DATA_BLOCK "MOD"   // DB57
// stored: InstanceOfName AFB_MODULES, InstanceOfType FB
"AFB_MODULES"
BEGIN
   ADIN[0].input := 536.3774;
   ADIN[0].monitorfault := TRUE;
   ADIN[0].p1s := FALSE;
   ADIN[0].p100ms := TRUE;
   ADIN[0].generalackn := FALSE;
   ADIN[0].reset := FALSE;
   ADIN[0].mute := FALSE;
   ADIN[0].Unit := WSTRING#'';
   ADIN[0].Switch := FALSE;
   ADIN[0].alarm_adin := FALSE;
   ADIN[0].plcackn_adin := FALSE;
   ADIN[0].siren_adin := FALSE;
   ADIN[0].hmiackn_adin := FALSE;
   ADIN[0].i."time".on_set := 0;
   ADIN[0].i."time".off_set := 0;
   ADIN[0].i."time".on_act := 0;
   ADIN[0].i."time".off_act := 0;
   ADIN[0].i.setup.comparison := 0;
   ADIN[0].i.setup.reference := 1900.0;
   ADIN[0].i.setup.alarm := FALSE;
   ADIN[0].i.setup.triggerversion := FALSE;
   ADIN[0].i.faults.adin.setup.en := FALSE;
   ADIN[0].i.faults.adin.setup.spon := 0.0;
   ADIN[0].i.faults.adin.don.countup := FALSE;
   ADIN[0].i.faults.adin.don.sp := 0;
   ADIN[0].i.faults.adin.don.actual := 0;
   ADIN[0].i.faults.adin.don.end := FALSE;
   ADIN[0].i.faults.adin.status.plcackn := FALSE;
   ADIN[0].i.faults.adin.status.alarm := FALSE;
   ADIN[0].i.faults.adin.status.siren := FALSE;
   ADIN[0].i.faults.fpreset := FALSE;
   ADIN[0].i.sim.cmdon := FALSE;
   ADIN[0].i.sim.cmdoff := FALSE;
   ADIN[0].i.sim.simulated := FALSE;
   ADIN[0].i.sim.cmdforce := FALSE;
   ADIN[0].i.sim.cmdunforce := FALSE;
   ADIN[0].i.sim.forced := FALSE;
   ADIN[0].i.status.rawinput := 525.5537;
   ADIN[0].i.status.processed := FALSE;
   ADIN[0].i.status.switch_active := FALSE;
   ADIN[0].i.status.alarm_monitor := FALSE;
   ADIN[0].i.status.fault := FALSE;
   ADIN[0].i.unit := WSTRING#'';
   // AIN[0] : LT44_01_01
   AIN[0].in := 12542;
   AIN[0].generalackn := FALSE;
   AIN[0].reset := FALSE;
   AIN[0].mute := FALSE;
   AIN[0].p1s := FALSE;
   AIN[0].p100ms := FALSE;
   AIN[0].t_sys := DTL#2025-10-07-08:40:00.150809;
   AIN[0]."type" := 2;
   AIN[0].output := 4.536314;
   AIN[0].i.chn."type" := 1;
   AIN[0].i.chn.in := 12534.0;
   AIN[0].i.chn.high := 27648.0;
   AIN[0].i.chn.low := 0.0;
   AIN[0].i.scale.high := 10.0;
   AIN[0].i.scale.low := 0.0;
   AIN[0].i.scale.factor := 1.0;
   AIN[0].i.scale.set := TRUE;
   AIN[0].i.sim.en := FALSE;
   AIN[0].i.sim.value := 0.0;
   AIN[0].i.exp.en := FALSE;
   AIN[0].i.exp.init := FALSE;
   AIN[0].i.exp.T := 0.0;
   AIN[0].i.exp.limit := 0.0;
   AIN[0].i.exp."dt" := 0.0;
   AIN[0].i.exp."a" := 0.0;
   AIN[0].i.faults.hh.setup.en := TRUE;
   AIN[0].i.faults.hh.setup.spon := 1.0;
   AIN[0].i.faults.hh.don.countup := FALSE;
   AIN[0].i.faults.hh.don.sp := 10;
   AIN[0].i.faults.hh.don.actual := 0;
   AIN[0].i.faults.hh.don.end := FALSE;
   AIN[0].i.faults.hh.status.plcackn := FALSE;
   AIN[0].i.faults.hh.status.alarm := FALSE;
   AIN[0].i.faults.hh.status.siren := FALSE;
   AIN[0].i.faults.h.setup.en := TRUE;
   AIN[0].i.faults.h.setup.spon := 10.0;
   AIN[0].i.faults.h.don.countup := FALSE;
   AIN[0].i.faults.h.don.sp := 100;
   AIN[0].i.faults.h.don.actual := 0;
   AIN[0].i.faults.h.don.end := FALSE;
   AIN[0].i.faults.h.status.plcackn := FALSE;
   AIN[0].i.faults.h.status.alarm := FALSE;
   AIN[0].i.faults.h.status.siren := FALSE;
   AIN[0].i.faults.l.setup.en := TRUE;
   AIN[0].i.faults.l.setup.spon := 0.0;
   AIN[0].i.faults.l.don.countup := FALSE;
   AIN[0].i.faults.l.don.sp := 0;
   AIN[0].i.faults.l.don.actual := 0;
   AIN[0].i.faults.l.don.end := FALSE;
   AIN[0].i.faults.l.status.plcackn := FALSE;
   AIN[0].i.faults.l.status.alarm := FALSE;
   AIN[0].i.faults.l.status.siren := FALSE;
   AIN[0].i.faults.ll.setup.en := TRUE;
   AIN[0].i.faults.ll.setup.spon := 0.0;
   AIN[0].i.faults.ll.don.countup := FALSE;
   AIN[0].i.faults.ll.don.sp := 0;
   AIN[0].i.faults.ll.don.actual := 0;
   AIN[0].i.faults.ll.don.end := FALSE;
   AIN[0].i.faults.ll.status.plcackn := FALSE;
   AIN[0].i.faults.ll.status.alarm := FALSE;
   AIN[0].i.faults.ll.status.siren := FALSE;
   AIN[0].i.faults.sp_hh := 5.6;
   AIN[0].i.faults.sp_h := 5.3;
   AIN[0].i.faults.sp_l := 0.5;
   AIN[0].i.faults.sp_ll := 0.2;
   AIN[0].i.faults.fpreset := FALSE;
   AIN[0].i.trendlow := -1.0;
   AIN[0].i.trendhigh := 12.0;
   AIN[0].i.scaled := 4.53342;
   AIN[0].i.output := 4.53342;
   AIN[0].i.unit := WSTRING#'m';
   AIN[0].exp.init := FALSE;
   AIN[0].exp.Sn := 4.536314;
   AIN[0].exp.Xn := 4.536314;
   AIN[0].exp.lim_up := 0.0;
   AIN[0].exp.lim_down := 0.0;
   AIN[0].exp.t_buf := DTL#2025-10-07-08:40:00.150809;
   AIN[0].exp.t_diff := FALSE;
   AIN[0].calc.scalespan := 10.0;
   AIN[0].calc.chnspan := 27648.0;
   AIN[0].calc.xmax := 27648.0;
   AIN[0].calc.xmin := 0.0;
   AIN[0].calc.ymax := 10.0;
   AIN[0].calc.ymin := 0.0;
   AIN[0].calc.x := 12542.0;
   AIN[0].calc.y := 4.536314;
   AIN[0].calc.sign := TRUE;
   AIN[0].calc.scale."type" := 0;
   AIN[0].calc.scale.in := 0.0;
   AIN[0].calc.scale.scalehigh := 0.0;
   AIN[0].calc.scale.scalelow := 0.0;
   AIN[0].calc.scale.channelhigh := 0.0;
   AIN[0].calc.scale.channellow := 0.0;
   AIN[0].calc.scale.factor := 0.0;
   AIN[0].calc.scale.calc1 := 0.0;
   AIN[0].calc.scale.span := 0.0;
   AIN[0].calc.scale.output := 0.0;
   AIN[0].lastob_si.EV_CLASS := 16#00;
   AIN[0].lastob_si.EV_NUM := 16#00;
   AIN[0].lastob_si.PRIORITY := 16#00;
   AIN[0].lastob_si.NUM := 16#00;
   AIN[0].lastob_si.TYP2_3 := 16#00;
   AIN[0].lastob_si.TYP1 := 16#00;
   AIN[0].lastob_si.ZI1 := 16#0000;
   AIN[0].lastob_si.ZI2_3 := 16#0000_0000;
   AIN[0].startob_si.EV_CLASS := 16#00;
   AIN[0].startob_si.EV_NUM := 16#00;
   AIN[0].startob_si.PRIORITY := 16#00;
   AIN[0].startob_si.NUM := 16#00;
   AIN[0].startob_si.TYP2_3 := 16#00;
   AIN[0].startob_si.TYP1 := 16#00;
   AIN[0].startob_si.ZI1 := 16#0000;
   AIN[0].startob_si.ZI2_3 := 16#0000_0000;
   AIN[0].err := 0;
   AIN[0].hilow := TRUE;
   AIN[0].factor := FALSE;
   DIFF[0].Minuend := 0.0;
   DIFF[0].Subtrahend := 0.0;
   DIFF[0].unit := WSTRING#'';
   DIFF[0].generalackn := FALSE;
   DIFF[0].reset := FALSE;
   DIFF[0].mute := FALSE;
   DIFF[0].p1s := FALSE;
   DIFF[0].p100ms := FALSE;
   DIFF[0].output := 0.0;
   DIFF[0].i.sim.en := FALSE;
   DIFF[0].i.sim.value := 0.0;
   DIFF[0].i.faults.hh.setup.en := FALSE;
   DIFF[0].i.faults.hh.setup.spon := 0.0;
   DIFF[0].i.faults.hh.don.countup := FALSE;
   DIFF[0].i.faults.hh.don.sp := 0;
   DIFF[0].i.faults.hh.don.actual := 0;
   DIFF[0].i.faults.hh.don.end := FALSE;
   DIFF[0].i.faults.hh.status.plcackn := FALSE;
   DIFF[0].i.faults.hh.status.alarm := FALSE;
   DIFF[0].i.faults.hh.status.siren := FALSE;
   DIFF[0].i.faults.h.setup.en := FALSE;
   DIFF[0].i.faults.h.setup.spon := 0.0;
   DIFF[0].i.faults.h.don.countup := FALSE;
   DIFF[0].i.faults.h.don.sp := 0;
   DIFF[0].i.faults.h.don.actual := 0;
   DIFF[0].i.faults.h.don.end := FALSE;
   DIFF[0].i.faults.h.status.plcackn := FALSE;
   DIFF[0].i.faults.h.status.alarm := FALSE;
   DIFF[0].i.faults.h.status.siren := FALSE;
   DIFF[0].i.faults.l.setup.en := FALSE;
   DIFF[0].i.faults.l.setup.spon := 0.0;
   DIFF[0].i.faults.l.don.countup := FALSE;
   DIFF[0].i.faults.l.don.sp := 0;
   DIFF[0].i.faults.l.don.actual := 0;
   DIFF[0].i.faults.l.don.end := FALSE;
   DIFF[0].i.faults.l.status.plcackn := FALSE;
   DIFF[0].i.faults.l.status.alarm := FALSE;
   DIFF[0].i.faults.l.status.siren := FALSE;
   DIFF[0].i.faults.ll.setup.en := FALSE;
   DIFF[0].i.faults.ll.setup.spon := 0.0;
   DIFF[0].i.faults.ll.don.countup := FALSE;
   DIFF[0].i.faults.ll.don.sp := 0;
   DIFF[0].i.faults.ll.don.actual := 0;
   DIFF[0].i.faults.ll.don.end := FALSE;
   DIFF[0].i.faults.ll.status.plcackn := FALSE;
   DIFF[0].i.faults.ll.status.alarm := FALSE;
   DIFF[0].i.faults.ll.status.siren := FALSE;
   DIFF[0].i.faults.sp_hh := 0.0;
   DIFF[0].i.faults.sp_h := 0.0;
   DIFF[0].i.faults.sp_l := 0.0;
   DIFF[0].i.faults.sp_ll := 0.0;
   DIFF[0].i.faults.fpreset := FALSE;
   DIFF[0].i.minuend := 0.0;
   DIFF[0].i.subtrahend := 0.0;
   DIFF[0].i.trendhigh := 0.0;
   DIFF[0].i.output := 0.0;
   DIFF[0].i.unit := WSTRING#'';
   // DIN[0] : LsH44_01_01
   DIN[0].input := TRUE;
   DIN[0].monitorfault := TRUE;
   DIN[0].p1s := FALSE;
   DIN[0].p100ms := FALSE;
   DIN[0].generalackn := FALSE;
   DIN[0].reset := FALSE;
   DIN[0].mute := FALSE;
   DIN[0].Switch := FALSE;
   DIN[0].alarm_din := FALSE;
   DIN[0].plcackn_din := FALSE;
   DIN[0].siren_din := FALSE;
   DIN[0].hmiackn_din := FALSE;
   DIN[0].i."time".on_set := 0;
   DIN[0].i."time".off_set := 0;
   DIN[0].i."time".on_act := 0;
   DIN[0].i."time".off_act := 0;
   DIN[0].i.setup.polarity := TRUE;
   DIN[0].i.setup.triggerversion := FALSE;
   DIN[0].i.faults.din.setup.en := FALSE;
   DIN[0].i.faults.din.setup.spon := 0.0;
   DIN[0].i.faults.din.don.countup := FALSE;
   DIN[0].i.faults.din.don.sp := 0;
   DIN[0].i.faults.din.don.actual := 0;
   DIN[0].i.faults.din.don.end := FALSE;
   DIN[0].i.faults.din.status.plcackn := FALSE;
   DIN[0].i.faults.din.status.alarm := FALSE;
   DIN[0].i.faults.din.status.siren := FALSE;
   DIN[0].i.faults.fpreset := FALSE;
   DIN[0].i.sim.cmdon := FALSE;
   DIN[0].i.sim.cmdoff := FALSE;
   DIN[0].i.sim.simulated := FALSE;
   DIN[0].i.sim.cmdforce := FALSE;
   DIN[0].i.sim.cmdunforce := FALSE;
   DIN[0].i.sim.forced := FALSE;
   DIN[0].i.status.rawinput := TRUE;
   DIN[0].i.status.processed := FALSE;
   DIN[0].i.status.switch_active := FALSE;
   DIN[0].i.status.alarm_monitor := FALSE;
   DIN[0].i.status.fault := FALSE;
   // MTR[0] : P44_05
   MTR[0].start := FALSE;
   MTR[0].spsource := FALSE;
   MTR[0].followup := FALSE;
   MTR[0].pidrun := TRUE;
   MTR[0].fb := FALSE;
   MTR[0].mcb := FALSE;
   MTR[0].ctrl := TRUE;
   MTR[0].vfdnotrip := FALSE;
   MTR[0].block := FALSE;
   MTR[0].generalackn := FALSE;
   MTR[0].reset := FALSE;
   MTR[0].mute := FALSE;
   MTR[0].autoset := FALSE;
   MTR[0].manualset := FALSE;
   MTR[0].p1s := FALSE;
   MTR[0].p100ms := FALSE;
   MTR[0].blink := TRUE;
   MTR[0].PV := 4.000289;
   MTR[0].PV_unit := WSTRING#'';
   MTR[0].EXT_SP := 0.0;
   MTR[0].FUP := 20.0;
   MTR[0].Out_unit := WSTRING#'';
   MTR[0].run := FALSE;
   MTR[0].vfb := FALSE;
   MTR[0].reference := 0;
   MTR[0].i.cmd.auto := FALSE;
   MTR[0].i.cmd.man := FALSE;
   MTR[0].i.cmd.start := FALSE;
   MTR[0].i.cmd.stop := FALSE;
   MTR[0].i.ind.auto := FALSE;
   MTR[0].i.ind.man := TRUE;
   MTR[0].i.ind.start := FALSE;
   MTR[0].i.ind.stop := TRUE;
   MTR[0].i.sim.fb := FALSE;
   MTR[0].i.sim.ctrl := FALSE;
   MTR[0].i.faults.ftr.setup.en := TRUE;
   MTR[0].i.faults.ftr.setup.spon := 6.0;
   MTR[0].i.faults.ftr.don.countup := FALSE;
   MTR[0].i.faults.ftr.don.sp := 60;
   MTR[0].i.faults.ftr.don.actual := 0;
   MTR[0].i.faults.ftr.don.end := FALSE;
   MTR[0].i.faults.ftr.status.plcackn := FALSE;
   MTR[0].i.faults.ftr.status.alarm := FALSE;
   MTR[0].i.faults.ftr.status.siren := FALSE;
   MTR[0].i.faults.fts.setup.en := TRUE;
   MTR[0].i.faults.fts.setup.spon := 6.0;
   MTR[0].i.faults.fts.don.countup := FALSE;
   MTR[0].i.faults.fts.don.sp := 60;
   MTR[0].i.faults.fts.don.actual := 0;
   MTR[0].i.faults.fts.don.end := FALSE;
   MTR[0].i.faults.fts.status.plcackn := FALSE;
   MTR[0].i.faults.fts.status.alarm := FALSE;
   MTR[0].i.faults.fts.status.siren := FALSE;
   MTR[0].i.faults.mcb.setup.en := FALSE;
   MTR[0].i.faults.mcb.setup.spon := 2.0;
   MTR[0].i.faults.mcb.don.countup := FALSE;
   MTR[0].i.faults.mcb.don.sp := 20;
   MTR[0].i.faults.mcb.don.actual := 0;
   MTR[0].i.faults.mcb.don.end := FALSE;
   MTR[0].i.faults.mcb.status.plcackn := FALSE;
   MTR[0].i.faults.mcb.status.alarm := FALSE;
   MTR[0].i.faults.mcb.status.siren := FALSE;
   MTR[0].i.faults.ctrl.setup.en := TRUE;
   MTR[0].i.faults.ctrl.setup.spon := 2.0;
   MTR[0].i.faults.ctrl.don.countup := FALSE;
   MTR[0].i.faults.ctrl.don.sp := 20;
   MTR[0].i.faults.ctrl.don.actual := 0;
   MTR[0].i.faults.ctrl.don.end := FALSE;
   MTR[0].i.faults.ctrl.status.plcackn := FALSE;
   MTR[0].i.faults.ctrl.status.alarm := FALSE;
   MTR[0].i.faults.ctrl.status.siren := FALSE;
   MTR[0].i.faults.vfd.setup.en := FALSE;
   MTR[0].i.faults.vfd.setup.spon := 5.0;
   MTR[0].i.faults.vfd.don.countup := FALSE;
   MTR[0].i.faults.vfd.don.sp := 50;
   MTR[0].i.faults.vfd.don.actual := 0;
   MTR[0].i.faults.vfd.don.end := FALSE;
   MTR[0].i.faults.vfd.status.plcackn := FALSE;
   MTR[0].i.faults.vfd.status.alarm := FALSE;
   MTR[0].i.faults.vfd.status.siren := FALSE;
   MTR[0].i.faults.il.setup.en := FALSE;
   MTR[0].i.faults.il.setup.spon := 0.0;
   MTR[0].i.faults.il.don.countup := FALSE;
   MTR[0].i.faults.il.don.sp := 0;
   MTR[0].i.faults.il.don.actual := 0;
   MTR[0].i.faults.il.don.end := FALSE;
   MTR[0].i.faults.il.status.plcackn := FALSE;
   MTR[0].i.faults.il.status.alarm := FALSE;
   MTR[0].i.faults.il.status.siren := FALSE;
   MTR[0].i.faults.fpreset := FALSE;
   MTR[0].i.pid.mode := FALSE;
   MTR[0].i.pid.action := TRUE;
   MTR[0].i.pid.spsource := FALSE;
   MTR[0].i.pid.followup := FALSE;
   MTR[0].i.pid.cmdrst := TRUE;
   MTR[0].i.pid.pidrun := TRUE;
   MTR[0].i.pid.P := 0.5;
   MTR[0].i.pid.I := 3;
   MTR[0].i.pid.D := 0;
   MTR[0].i.pid.SP := 4.0;
   MTR[0].i.pid.PV := 3.996672;
   MTR[0].i.pid.OFFVAL := 0.0;
   MTR[0].i.pid.LMN := 0.0;
   MTR[0].i.pid.OP := 0.0;
   MTR[0].i.pid.L := 10.0;
   MTR[0].i.pid.H := 100.0;
   MTR[0].i.pid.EXT_SP := 0.0;
   MTR[0].i.pid.FUP := 20.0;
   MTR[0].i.pid.ITLVAL := 70.0;
   MTR[0].i.pid.pvunit := WSTRING#'';
   MTR[0].i.pid.outunit := WSTRING#'%';
   MTR[0].i.pid.init.req := TRUE;
   MTR[0].i.pid.init.dur := 15.0;
   MTR[0].i.pid.init.delay.in.spon := 0.0;
   MTR[0].i.pid.init.delay.don.trigger := FALSE;
   MTR[0].i.pid.init.delay.don.sp := 0;
   MTR[0].i.pid.init.delay.don.actual := 0;
   MTR[0].i.pid.init.delay.don.end := FALSE;
   MTR[0].i.pid.init.delay.out.on := FALSE;
   MTR[0].i.unscale.in := 0.0;
   MTR[0].i.unscale.inhigh := 100.0;
   MTR[0].i.unscale.inlow := 0.0;
   MTR[0].i.unscale.outhigh := 27648.0;
   MTR[0].i.unscale.outlow := 0.0;
   MTR[0].i.unscale.output := 0.0;
   MTR[0].i.unscale.set := TRUE;
   MTR[0].i.arh.checkafter := 0;
   MTR[0].i.arh.lastmaint := 0;
   MTR[0].i.arh.difference := 4;
   MTR[0].i.arh.actual := 4;
   MTR[0].i.arh.seconds := 686;
   MTR[0].i.arh.hour := FALSE;
   MTR[0].i.arh.resetarh := FALSE;
   MTR[0].i.arh.enable := FALSE;
   MTR[0].i.arh.maintenance := FALSE;
   MTR[0].i.arh.completed := FALSE;
   MTR[0].i.status.vfb := FALSE;
   MTR[0].i.status.vctrl := TRUE;
   MTR[0].i.status.ilstart := TRUE;
   MTR[0].i.status.fault := FALSE;
   MTR[0].i.status.maint := FALSE;
   MTR[0].i.status.icon := 0;
   MTR[0].i.delay.in.spon := 0.0;
   MTR[0].i.delay.in.spoff := 0.0;
   MTR[0].i.delay.don.trigger := FALSE;
   MTR[0].i.delay.don.sp := 0;
   MTR[0].i.delay.don.actual := 0;
   MTR[0].i.delay.don.end := FALSE;
   MTR[0].i.delay.doff.trigger := FALSE;
   MTR[0].i.delay.doff.sp := 0;
   MTR[0].i.delay.doff.actual := 0;
   MTR[0].i.delay.doff.end := FALSE;
   MTR[0].i.delay.out.on := FALSE;
   MTR[0].i.out.manrun := FALSE;
   MTR[0].i.out.run := FALSE;
   MTR[0].i.out.ref := 0;
   MTR[0].cont.COM_RST := TRUE;
   MTR[0].cont.MAN_ON := FALSE;
   MTR[0].cont.SP_INT := 4.0;
   MTR[0].cont.PV_IN := 4.000289;
   MTR[0].cont.GAIN := 0.5;
   MTR[0].cont.TI := T#3MS;
   MTR[0].cont.TD := T#0MS;
   MTR[0].cont.LMN_HLM := 100.0;
   MTR[0].cont.LMN_LLM := 10.0;
   MTR[0].cont.LMN_FAC := 1.0;
   MTR[0].cont.LMN_OFF := 0.0;
   MTR[0].cont.I_ITLVAL := 0.0;
   MTR[0].cont.LMN := 0.0;
   MTR[0].calc.inspan := 100.0;
   MTR[0].calc.outspan := 27648.0;
   MTR[0].calc.xmax := 100.0;
   MTR[0].calc.xmin := 0.0;
   MTR[0].calc.ymax := 27648.0;
   MTR[0].calc.ymin := 0.0;
   MTR[0].calc.x := 0.0;
   MTR[0].calc.y := 0.0;
   MTR[0].calc.sign := TRUE;
   MTRLIN[0].start := FALSE;
   MTRLIN[0].followup := FALSE;
   MTRLIN[0].fb := TRUE;
   MTRLIN[0].mcb := TRUE;
   MTRLIN[0].ctrl := FALSE;
   MTRLIN[0].vfdnotrip := TRUE;
   MTRLIN[0].block := FALSE;
   MTRLIN[0].generalackn := FALSE;
   MTRLIN[0].reset := FALSE;
   MTRLIN[0].mute := FALSE;
   MTRLIN[0].autoset := FALSE;
   MTRLIN[0].manualset := FALSE;
   MTRLIN[0].p1s := FALSE;
   MTRLIN[0].p100ms := TRUE;
   MTRLIN[0].blink := TRUE;
   MTRLIN[0].PV := 0.0;
   MTRLIN[0].PV_unit := WSTRING#'°C';
   MTRLIN[0].FUP := 0.0;
   MTRLIN[0].Out_unit := WSTRING#'';
   MTRLIN[0].run := FALSE;
   MTRLIN[0].vfb := TRUE;
   MTRLIN[0].reference := 0;
   MTRLIN[0].i.cmd.auto := FALSE;
   MTRLIN[0].i.cmd.man := FALSE;
   MTRLIN[0].i.cmd.start := FALSE;
   MTRLIN[0].i.cmd.stop := FALSE;
   MTRLIN[0].i.ind.auto := FALSE;
   MTRLIN[0].i.ind.man := TRUE;
   MTRLIN[0].i.ind.start := FALSE;
   MTRLIN[0].i.ind.stop := TRUE;
   MTRLIN[0].i.sim.fb := FALSE;
   MTRLIN[0].i.sim.ctrl := FALSE;
   MTRLIN[0].i.faults.ftr.setup.en := TRUE;
   MTRLIN[0].i.faults.ftr.setup.spon := 5.0;
   MTRLIN[0].i.faults.ftr.don.countup := FALSE;
   MTRLIN[0].i.faults.ftr.don.sp := 50;
   MTRLIN[0].i.faults.ftr.don.actual := 0;
   MTRLIN[0].i.faults.ftr.don.end := FALSE;
   MTRLIN[0].i.faults.ftr.status.plcackn := FALSE;
   MTRLIN[0].i.faults.ftr.status.alarm := FALSE;
   MTRLIN[0].i.faults.ftr.status.siren := FALSE;
   MTRLIN[0].i.faults.fts.setup.en := TRUE;
   MTRLIN[0].i.faults.fts.setup.spon := 5.0;
   MTRLIN[0].i.faults.fts.don.countup := FALSE;
   MTRLIN[0].i.faults.fts.don.sp := 50;
   MTRLIN[0].i.faults.fts.don.actual := 0;
   MTRLIN[0].i.faults.fts.don.end := FALSE;
   MTRLIN[0].i.faults.fts.status.plcackn := FALSE;
   MTRLIN[0].i.faults.fts.status.alarm := FALSE;
   MTRLIN[0].i.faults.fts.status.siren := FALSE;
   MTRLIN[0].i.faults.mcb.setup.en := TRUE;
   MTRLIN[0].i.faults.mcb.setup.spon := 1.0;
   MTRLIN[0].i.faults.mcb.don.countup := FALSE;
   MTRLIN[0].i.faults.mcb.don.sp := 10;
   MTRLIN[0].i.faults.mcb.don.actual := 0;
   MTRLIN[0].i.faults.mcb.don.end := FALSE;
   MTRLIN[0].i.faults.mcb.status.plcackn := FALSE;
   MTRLIN[0].i.faults.mcb.status.alarm := FALSE;
   MTRLIN[0].i.faults.mcb.status.siren := FALSE;
   MTRLIN[0].i.faults.ctrl.setup.en := TRUE;
   MTRLIN[0].i.faults.ctrl.setup.spon := 1.0;
   MTRLIN[0].i.faults.ctrl.don.countup := FALSE;
   MTRLIN[0].i.faults.ctrl.don.sp := 10;
   MTRLIN[0].i.faults.ctrl.don.actual := 0;
   MTRLIN[0].i.faults.ctrl.don.end := FALSE;
   MTRLIN[0].i.faults.ctrl.status.plcackn := FALSE;
   MTRLIN[0].i.faults.ctrl.status.alarm := FALSE;
   MTRLIN[0].i.faults.ctrl.status.siren := FALSE;
   MTRLIN[0].i.faults.vfd.setup.en := TRUE;
   MTRLIN[0].i.faults.vfd.setup.spon := 1.0;
   MTRLIN[0].i.faults.vfd.don.countup := FALSE;
   MTRLIN[0].i.faults.vfd.don.sp := 10;
   MTRLIN[0].i.faults.vfd.don.actual := 0;
   MTRLIN[0].i.faults.vfd.don.end := FALSE;
   MTRLIN[0].i.faults.vfd.status.plcackn := FALSE;
   MTRLIN[0].i.faults.vfd.status.alarm := TRUE;
   MTRLIN[0].i.faults.vfd.status.siren := TRUE;
   MTRLIN[0].i.faults.il.setup.en := FALSE;
   MTRLIN[0].i.faults.il.setup.spon := 0.0;
   MTRLIN[0].i.faults.il.don.countup := FALSE;
   MTRLIN[0].i.faults.il.don.sp := 0;
   MTRLIN[0].i.faults.il.don.actual := 0;
   MTRLIN[0].i.faults.il.don.end := FALSE;
   MTRLIN[0].i.faults.il.status.plcackn := FALSE;
   MTRLIN[0].i.faults.il.status.alarm := FALSE;
   MTRLIN[0].i.faults.il.status.siren := FALSE;
   MTRLIN[0].i.faults.fpreset := FALSE;
   MTRLIN[0].i.scale.in := 0.0;
   MTRLIN[0].i.scale.instart := 0.0;
   MTRLIN[0].i.scale.inend := 0.0;
   MTRLIN[0].i.scale.outstart := 0.0;
   MTRLIN[0].i.scale.outend := 0.0;
   MTRLIN[0].i.scale.output := 0.0;
   MTRLIN[0].i.scale.set := FALSE;
   MTRLIN[0].i.ctrl.mode := TRUE;
   MTRLIN[0].i.ctrl.linear := FALSE;
   MTRLIN[0].i.ctrl.PV := 0.0;
   MTRLIN[0].i.ctrl.OFFVAL := 0.0;
   MTRLIN[0].i.ctrl.OP := 100.0;
   MTRLIN[0].i.ctrl.FUP := 0.0;
   MTRLIN[0].i.ctrl.ITLVAL := 0.0;
   MTRLIN[0].i.ctrl.pvunit := WSTRING#'°C';
   MTRLIN[0].i.ctrl.outunit := WSTRING#'%';
   MTRLIN[0].i.ctrl.init.req := FALSE;
   MTRLIN[0].i.ctrl.init.dur := 0.0;
   MTRLIN[0].i.ctrl.init.delay.in.spon := 0.0;
   MTRLIN[0].i.ctrl.init.delay.don.trigger := FALSE;
   MTRLIN[0].i.ctrl.init.delay.don.sp := 0;
   MTRLIN[0].i.ctrl.init.delay.don.actual := 0;
   MTRLIN[0].i.ctrl.init.delay.don.end := FALSE;
   MTRLIN[0].i.ctrl.init.delay.out.on := FALSE;
   MTRLIN[0].i.unscale.in := 100.0;
   MTRLIN[0].i.unscale.inhigh := 100.0;
   MTRLIN[0].i.unscale.inlow := 0.0;
   MTRLIN[0].i.unscale.outhigh := 1370.0;
   MTRLIN[0].i.unscale.outlow := 0.0;
   MTRLIN[0].i.unscale.output := 1370.0;
   MTRLIN[0].i.unscale.set := TRUE;
   MTRLIN[0].i.arh.checkafter := 0;
   MTRLIN[0].i.arh.lastmaint := 0;
   MTRLIN[0].i.arh.difference := 7;
   MTRLIN[0].i.arh.actual := 7;
   MTRLIN[0].i.arh.seconds := 2414;
   MTRLIN[0].i.arh.hour := FALSE;
   MTRLIN[0].i.arh.resetarh := FALSE;
   MTRLIN[0].i.arh.enable := FALSE;
   MTRLIN[0].i.arh.maintenance := FALSE;
   MTRLIN[0].i.arh.completed := FALSE;
   MTRLIN[0].i.status.vfb := TRUE;
   MTRLIN[0].i.status.vctrl := FALSE;
   MTRLIN[0].i.status.ilstart := FALSE;
   MTRLIN[0].i.status.fault := TRUE;
   MTRLIN[0].i.status.maint := FALSE;
   MTRLIN[0].i.status.icon := 0;
   MTRLIN[0].i.delay.in.spon := 0.0;
   MTRLIN[0].i.delay.in.spoff := 0.0;
   MTRLIN[0].i.delay.don.trigger := FALSE;
   MTRLIN[0].i.delay.don.sp := 0;
   MTRLIN[0].i.delay.don.actual := 0;
   MTRLIN[0].i.delay.don.end := FALSE;
   MTRLIN[0].i.delay.doff.trigger := FALSE;
   MTRLIN[0].i.delay.doff.sp := 0;
   MTRLIN[0].i.delay.doff.actual := 0;
   MTRLIN[0].i.delay.doff.end := FALSE;
   MTRLIN[0].i.delay.out.on := FALSE;
   MTRLIN[0].i.out.manrun := FALSE;
   MTRLIN[0].i.out.run := FALSE;
   MTRLIN[0].i.out.ref := 1370;
   MTRLIN[0].calc.inspan := 100.0;
   MTRLIN[0].calc.outspan := 1370.0;
   MTRLIN[0].calc.xmax := 100.0;
   MTRLIN[0].calc.xmin := 0.0;
   MTRLIN[0].calc.ymax := 1370.0;
   MTRLIN[0].calc.ymin := 0.0;
   MTRLIN[0].calc.x := 100.0;
   MTRLIN[0].calc.y := 1370.0;
   MTRLIN[0].calc.speedmin := 0.0;
   MTRLIN[0].calc.speedmax := 100.0;
   MTRLIN[0].calc.sign := TRUE;
   // MTRDIR[0] : P44_01
   MTRDIR[0].start := FALSE;
   MTRDIR[0].fb := FALSE;
   MTRDIR[0].mcb := TRUE;
   MTRDIR[0].ctrl := TRUE;
   MTRDIR[0].block := FALSE;
   MTRDIR[0].generalackn := FALSE;
   MTRDIR[0].reset := FALSE;
   MTRDIR[0].mute := FALSE;
   MTRDIR[0].autoset := FALSE;
   MTRDIR[0].manualset := FALSE;
   MTRDIR[0].p1s := FALSE;
   MTRDIR[0].p100ms := FALSE;
   MTRDIR[0].blink := TRUE;
   MTRDIR[0].run := FALSE;
   MTRDIR[0].vfb := FALSE;
   MTRDIR[0].i.cmd.auto := FALSE;
   MTRDIR[0].i.cmd.man := FALSE;
   MTRDIR[0].i.cmd.start := FALSE;
   MTRDIR[0].i.cmd.stop := FALSE;
   MTRDIR[0].i.ind.auto := FALSE;
   MTRDIR[0].i.ind.man := TRUE;
   MTRDIR[0].i.ind.start := FALSE;
   MTRDIR[0].i.ind.stop := TRUE;
   MTRDIR[0].i.sim.fb := FALSE;
   MTRDIR[0].i.sim.ctrl := FALSE;
   MTRDIR[0].i.faults.ftr.setup.en := TRUE;
   MTRDIR[0].i.faults.ftr.setup.spon := 130.0;
   MTRDIR[0].i.faults.ftr.don.countup := FALSE;
   MTRDIR[0].i.faults.ftr.don.sp := 1300;
   MTRDIR[0].i.faults.ftr.don.actual := 0;
   MTRDIR[0].i.faults.ftr.don.end := FALSE;
   MTRDIR[0].i.faults.ftr.status.plcackn := FALSE;
   MTRDIR[0].i.faults.ftr.status.alarm := FALSE;
   MTRDIR[0].i.faults.ftr.status.siren := FALSE;
   MTRDIR[0].i.faults.fts.setup.en := TRUE;
   MTRDIR[0].i.faults.fts.setup.spon := 6.0;
   MTRDIR[0].i.faults.fts.don.countup := FALSE;
   MTRDIR[0].i.faults.fts.don.sp := 60;
   MTRDIR[0].i.faults.fts.don.actual := 0;
   MTRDIR[0].i.faults.fts.don.end := FALSE;
   MTRDIR[0].i.faults.fts.status.plcackn := FALSE;
   MTRDIR[0].i.faults.fts.status.alarm := FALSE;
   MTRDIR[0].i.faults.fts.status.siren := FALSE;
   MTRDIR[0].i.faults.mcb.setup.en := TRUE;
   MTRDIR[0].i.faults.mcb.setup.spon := 2.0;
   MTRDIR[0].i.faults.mcb.don.countup := FALSE;
   MTRDIR[0].i.faults.mcb.don.sp := 20;
   MTRDIR[0].i.faults.mcb.don.actual := 0;
   MTRDIR[0].i.faults.mcb.don.end := FALSE;
   MTRDIR[0].i.faults.mcb.status.plcackn := FALSE;
   MTRDIR[0].i.faults.mcb.status.alarm := FALSE;
   MTRDIR[0].i.faults.mcb.status.siren := FALSE;
   MTRDIR[0].i.faults.ctrl.setup.en := TRUE;
   MTRDIR[0].i.faults.ctrl.setup.spon := 2.0;
   MTRDIR[0].i.faults.ctrl.don.countup := FALSE;
   MTRDIR[0].i.faults.ctrl.don.sp := 20;
   MTRDIR[0].i.faults.ctrl.don.actual := 0;
   MTRDIR[0].i.faults.ctrl.don.end := FALSE;
   MTRDIR[0].i.faults.ctrl.status.plcackn := FALSE;
   MTRDIR[0].i.faults.ctrl.status.alarm := FALSE;
   MTRDIR[0].i.faults.ctrl.status.siren := FALSE;
   MTRDIR[0].i.faults.il.setup.en := FALSE;
   MTRDIR[0].i.faults.il.setup.spon := 0.0;
   MTRDIR[0].i.faults.il.don.countup := FALSE;
   MTRDIR[0].i.faults.il.don.sp := 0;
   MTRDIR[0].i.faults.il.don.actual := 0;
   MTRDIR[0].i.faults.il.don.end := FALSE;
   MTRDIR[0].i.faults.il.status.plcackn := FALSE;
   MTRDIR[0].i.faults.il.status.alarm := FALSE;
   MTRDIR[0].i.faults.il.status.siren := FALSE;
   MTRDIR[0].i.faults.fpreset := FALSE;
   MTRDIR[0].i.arh.checkafter := 0;
   MTRDIR[0].i.arh.lastmaint := 0;
   MTRDIR[0].i.arh.difference := 146;
   MTRDIR[0].i.arh.actual := 146;
   MTRDIR[0].i.arh.seconds := 796;
   MTRDIR[0].i.arh.hour := FALSE;
   MTRDIR[0].i.arh.resetarh := FALSE;
   MTRDIR[0].i.arh.enable := FALSE;
   MTRDIR[0].i.arh.maintenance := FALSE;
   MTRDIR[0].i.arh.completed := FALSE;
   MTRDIR[0].i.status.vfb := FALSE;
   MTRDIR[0].i.status.vctrl := TRUE;
   MTRDIR[0].i.status.ilstart := TRUE;
   MTRDIR[0].i.status.fault := FALSE;
   MTRDIR[0].i.status.maint := FALSE;
   MTRDIR[0].i.status.icon := 0;
   MTRDIR[0].i.delay.in.spon := 0.0;
   MTRDIR[0].i.delay.in.spoff := 0.0;
   MTRDIR[0].i.delay.don.trigger := FALSE;
   MTRDIR[0].i.delay.don.sp := 0;
   MTRDIR[0].i.delay.don.actual := 0;
   MTRDIR[0].i.delay.don.end := FALSE;
   MTRDIR[0].i.delay.doff.trigger := FALSE;
   MTRDIR[0].i.delay.doff.sp := 0;
   MTRDIR[0].i.delay.doff.actual := 0;
   MTRDIR[0].i.delay.doff.end := FALSE;
   MTRDIR[0].i.delay.out.on := FALSE;
   MTRDIR[0].i.out.manrun := FALSE;
   MTRDIR[0].i.out.run := FALSE;
   // VLV[0] : V04_01
   VLV[0].actmain := FALSE;
   VLV[0].actupper := FALSE;
   VLV[0].actlower := FALSE;
   VLV[0].fbmain := FALSE;
   VLV[0].fbupper := FALSE;
   VLV[0].fblower := FALSE;
   VLV[0].fbdeact := TRUE;
   VLV[0].blockmain := FALSE;
   VLV[0].blockupper := FALSE;
   VLV[0].blocklower := FALSE;
   VLV[0].generalackn := FALSE;
   VLV[0].reset := FALSE;
   VLV[0].mute := FALSE;
   VLV[0].autoset := FALSE;
   VLV[0].manualset := FALSE;
   VLV[0].p1s := TRUE;
   VLV[0].p100ms := FALSE;
   VLV[0].blink := TRUE;
   VLV[0]."type" := 0;
   VLV[0].main := FALSE;
   VLV[0].upper := FALSE;
   VLV[0].lower := FALSE;
   VLV[0].vfbmain := FALSE;
   VLV[0].vfbupper := FALSE;
   VLV[0].vfblower := FALSE;
   VLV[0].vfbdeact := TRUE;
   VLV[0].i.cmd.auto := FALSE;
   VLV[0].i.cmd.man := FALSE;
   VLV[0].i.cmd.main := FALSE;
   VLV[0].i.cmd.upper := FALSE;
   VLV[0].i.cmd.lower := FALSE;
   VLV[0].i.cmd.deact := FALSE;
   VLV[0].i.ind.auto := TRUE;
   VLV[0].i.ind.man := FALSE;
   VLV[0].i.ind.main := FALSE;
   VLV[0].i.ind.upper := FALSE;
   VLV[0].i.ind.lower := FALSE;
   VLV[0].i.ind.deact := FALSE;
   VLV[0].i.man.main := FALSE;
   VLV[0].i.man.upper := FALSE;
   VLV[0].i.man.lower := FALSE;
   VLV[0].i.sim.main := FALSE;
   VLV[0].i.sim.upper := FALSE;
   VLV[0].i.sim.lower := FALSE;
   VLV[0].i.sim.deact := FALSE;
   VLV[0].i.faults.ftamain.setup.en := TRUE;
   VLV[0].i.faults.ftamain.setup.spon := 6.0;
   VLV[0].i.faults.ftamain.don.countup := FALSE;
   VLV[0].i.faults.ftamain.don.sp := 60;
   VLV[0].i.faults.ftamain.don.actual := 0;
   VLV[0].i.faults.ftamain.don.end := FALSE;
   VLV[0].i.faults.ftamain.status.plcackn := FALSE;
   VLV[0].i.faults.ftamain.status.alarm := FALSE;
   VLV[0].i.faults.ftamain.status.siren := FALSE;
   VLV[0].i.faults.ftaupper.setup.en := FALSE;
   VLV[0].i.faults.ftaupper.setup.spon := 0.0;
   VLV[0].i.faults.ftaupper.don.countup := FALSE;
   VLV[0].i.faults.ftaupper.don.sp := 0;
   VLV[0].i.faults.ftaupper.don.actual := 0;
   VLV[0].i.faults.ftaupper.don.end := FALSE;
   VLV[0].i.faults.ftaupper.status.plcackn := FALSE;
   VLV[0].i.faults.ftaupper.status.alarm := FALSE;
   VLV[0].i.faults.ftaupper.status.siren := FALSE;
   VLV[0].i.faults.ftalower.setup.en := FALSE;
   VLV[0].i.faults.ftalower.setup.spon := 0.0;
   VLV[0].i.faults.ftalower.don.countup := FALSE;
   VLV[0].i.faults.ftalower.don.sp := 0;
   VLV[0].i.faults.ftalower.don.actual := 0;
   VLV[0].i.faults.ftalower.don.end := FALSE;
   VLV[0].i.faults.ftalower.status.plcackn := FALSE;
   VLV[0].i.faults.ftalower.status.alarm := FALSE;
   VLV[0].i.faults.ftalower.status.siren := FALSE;
   VLV[0].i.faults.ftd.setup.en := TRUE;
   VLV[0].i.faults.ftd.setup.spon := 6.0;
   VLV[0].i.faults.ftd.don.countup := FALSE;
   VLV[0].i.faults.ftd.don.sp := 60;
   VLV[0].i.faults.ftd.don.actual := 0;
   VLV[0].i.faults.ftd.don.end := FALSE;
   VLV[0].i.faults.ftd.status.plcackn := FALSE;
   VLV[0].i.faults.ftd.status.alarm := FALSE;
   VLV[0].i.faults.ftd.status.siren := FALSE;
   VLV[0].i.faults.il.setup.en := FALSE;
   VLV[0].i.faults.il.setup.spon := 0.0;
   VLV[0].i.faults.il.don.countup := FALSE;
   VLV[0].i.faults.il.don.sp := 0;
   VLV[0].i.faults.il.don.actual := 0;
   VLV[0].i.faults.il.don.end := FALSE;
   VLV[0].i.faults.il.status.plcackn := FALSE;
   VLV[0].i.faults.il.status.alarm := FALSE;
   VLV[0].i.faults.il.status.siren := FALSE;
   VLV[0].i.faults.fpreset := FALSE;
   VLV[0].i.delaymain.in.spon := 0.0;
   VLV[0].i.delaymain.in.spoff := 0.0;
   VLV[0].i.delaymain.don.trigger := FALSE;
   VLV[0].i.delaymain.don.sp := 0;
   VLV[0].i.delaymain.don.actual := 0;
   VLV[0].i.delaymain.don.end := FALSE;
   VLV[0].i.delaymain.doff.trigger := FALSE;
   VLV[0].i.delaymain.doff.sp := 0;
   VLV[0].i.delaymain.doff.actual := 0;
   VLV[0].i.delaymain.doff.end := FALSE;
   VLV[0].i.delaymain.out.on := FALSE;
   VLV[0].i.delayupper.in.spon := 0.0;
   VLV[0].i.delayupper.in.spoff := 0.0;
   VLV[0].i.delayupper.don.trigger := FALSE;
   VLV[0].i.delayupper.don.sp := 0;
   VLV[0].i.delayupper.don.actual := 0;
   VLV[0].i.delayupper.don.end := FALSE;
   VLV[0].i.delayupper.doff.trigger := FALSE;
   VLV[0].i.delayupper.doff.sp := 0;
   VLV[0].i.delayupper.doff.actual := 0;
   VLV[0].i.delayupper.doff.end := FALSE;
   VLV[0].i.delayupper.out.on := FALSE;
   VLV[0].i.delaylower.in.spon := 0.0;
   VLV[0].i.delaylower.in.spoff := 0.0;
   VLV[0].i.delaylower.don.trigger := FALSE;
   VLV[0].i.delaylower.don.sp := 0;
   VLV[0].i.delaylower.don.actual := 0;
   VLV[0].i.delaylower.don.end := FALSE;
   VLV[0].i.delaylower.doff.trigger := FALSE;
   VLV[0].i.delaylower.doff.sp := 0;
   VLV[0].i.delaylower.doff.actual := 0;
   VLV[0].i.delaylower.doff.end := FALSE;
   VLV[0].i.delaylower.out.on := FALSE;
   VLV[0].i.out.actmain := FALSE;
   VLV[0].i.out.actupper := FALSE;
   VLV[0].i.out.actlower := FALSE;
   VLV[0].i.status.vfbmain := FALSE;
   VLV[0].i.status.vfbupper := FALSE;
   VLV[0].i.status.vfblower := FALSE;
   VLV[0].i.status.vfbdeact := TRUE;
   VLV[0].i.status.fault := FALSE;
   VLV[0].i.status.ilactmain := TRUE;
   VLV[0].i.status.ilactupper := TRUE;
   VLV[0].i.status.ilactlower := TRUE;
   VLV[0].i.status.icon := 0;
   CVLV[0].control := FALSE;
   CVLV[0].spsource := FALSE;
   CVLV[0].followup := TRUE;
   CVLV[0].pidrun := TRUE;
   CVLV[0].block := FALSE;
   CVLV[0].p1s := FALSE;
   CVLV[0].p100ms := FALSE;
   CVLV[0].blink := TRUE;
   CVLV[0].PV := 0.0;
   CVLV[0].PV_unit := WSTRING#'';
   CVLV[0].EXT_SP := 0.0;
   CVLV[0].FUP := 0.0;
   CVLV[0].Out_unit := WSTRING#'%';
   CVLV[0].reference := 0;
   CVLV[0].i.pid.mode := FALSE;
   CVLV[0].i.pid.action := FALSE;
   CVLV[0].i.pid.spsource := FALSE;
   CVLV[0].i.pid.followup := TRUE;
   CVLV[0].i.pid.cmdrst := TRUE;
   CVLV[0].i.pid.pidrun := TRUE;
   CVLV[0].i.pid.P := 0.0;
   CVLV[0].i.pid.I := 0;
   CVLV[0].i.pid.D := 0;
   CVLV[0].i.pid.SP := 1729.0;
   CVLV[0].i.pid.PV := 0.0;
   CVLV[0].i.pid.OFFVAL := 0.0;
   CVLV[0].i.pid.LMN := 0.0;
   CVLV[0].i.pid.OP := 0.0;
   CVLV[0].i.pid.L := 0.0;
   CVLV[0].i.pid.H := 0.0;
   CVLV[0].i.pid.EXT_SP := 0.0;
   CVLV[0].i.pid.FUP := 0.0;
   CVLV[0].i.pid.ITLVAL := 0.0;
   CVLV[0].i.pid.pvunit := WSTRING#'';
   CVLV[0].i.pid.outunit := WSTRING#'%';
   CVLV[0].i.pid.init.req := FALSE;
   CVLV[0].i.pid.init.dur := 0.0;
   CVLV[0].i.pid.init.delay.in.spon := 0.0;
   CVLV[0].i.pid.init.delay.don.trigger := FALSE;
   CVLV[0].i.pid.init.delay.don.sp := 0;
   CVLV[0].i.pid.init.delay.don.actual := 0;
   CVLV[0].i.pid.init.delay.don.end := FALSE;
   CVLV[0].i.pid.init.delay.out.on := FALSE;
   CVLV[0].i.unscale.in := 0.0;
   CVLV[0].i.unscale.inhigh := 100.0;
   CVLV[0].i.unscale.inlow := 0.0;
   CVLV[0].i.unscale.outhigh := 20000.0;
   CVLV[0].i.unscale.outlow := 4000.0;
   CVLV[0].i.unscale.output := 4000.0;
   CVLV[0].i.unscale.set := TRUE;
   CVLV[0].i.status.ilstart := TRUE;
   CVLV[0].i.status.icon := 0;
   CVLV[0].i.out.ref := 4000;
   CVLV[0].i.out.control := FALSE;
   CVLV[0].i.out.vfbact := FALSE;
   CVLV[0].i.out.vfbdeact := TRUE;
   CVLV[0].cont.COM_RST := TRUE;
   CVLV[0].cont.MAN_ON := FALSE;
   CVLV[0].cont.SP_INT := 1729.0;
   CVLV[0].cont.PV_IN := 0.0;
   CVLV[0].cont.GAIN := 0.0;
   CVLV[0].cont.TI := T#0MS;
   CVLV[0].cont.TD := T#0MS;
   CVLV[0].cont.LMN_HLM := 0.0;
   CVLV[0].cont.LMN_LLM := 0.0;
   CVLV[0].cont.LMN_FAC := 1.0;
   CVLV[0].cont.LMN_OFF := 0.0;
   CVLV[0].cont.I_ITLVAL := 0.0;
   CVLV[0].cont.LMN := 0.0;
   CVLV[0].calc.inspan := 100.0;
   CVLV[0].calc.outspan := 16000.0;
   CVLV[0].calc.xmax := 100.0;
   CVLV[0].calc.xmin := 0.0;
   CVLV[0].calc.ymax := 20000.0;
   CVLV[0].calc.ymin := 4000.0;
   CVLV[0].calc.x := 0.0;
   CVLV[0].calc.y := 4000.0;
   CVLV[0].calc.sign := TRUE;
END_DATA_BLOCK

DATA_BLOCK "GET_DB"   // DB7
// stored: InstanceOfName GET_SFB, OfSystemLibElement GET, OfSystemLibVersion 1.3
"GET_SFB"
   // VAR_INPUT
   //    REQ : Bool;
   //    ID : Word;
   // END_VAR
   // VAR_OUTPUT
   //    NDR : Bool;
   //    ERROR : Bool;
   //    STATUS : Word;
   // END_VAR
   // VAR_IN_OUT
   //    ADDR_1 : Remote;
   //    ADDR_2 : Remote;
   //    ADDR_3 : Remote;
   //    ADDR_4 : Remote;
   //    RD_1 : Variant;
   //    RD_2 : Variant;
   //    RD_3 : Variant;
   //    RD_4 : Variant;
   // END_VAR
BEGIN
END_DATA_BLOCK

DATA_BLOCK "iPALARMS"   // DB500
AUTHOR : CH
FAMILY : Aktina
NAME : Faults
// stored: AutoNumber false, InstanceOfName pALARMS, InstanceOfType FB
"pALARMS"
BEGIN
   "75sf1".trigger := FALSE;
   "75sf1".release := TRUE;
   "75sf1".ctrlpoint := TRUE;
   "75sf1".enackn := TRUE;
   "75sf1".ensiren := TRUE;
   "75sf1".p100ms := TRUE;
   "75sf1".generalackn := FALSE;
   "75sf1".reset := FALSE;
   "75sf1".mute := FALSE;
   "75sf1".delay := 0.5;
   "75sf1".plcackn := FALSE;
   "75sf1".alarm := FALSE;
   "75sf1".siren := FALSE;
   "75sf1".hmiackn := FALSE;
   "75sf1".i.setup.en := TRUE;
   "75sf1".i.setup.spon := 0.0;
   "75sf1".i.don.countup := FALSE;
   "75sf1".i.don.sp := 5;
   "75sf1".i.don.actual := 0;
   "75sf1".i.don.end := FALSE;
   "75sf1".i.status.plcackn := FALSE;
   "75sf1".i.status.alarm := FALSE;
   "75sf1".i.status.siren := FALSE;
END_DATA_BLOCK
